FUNCTION REPLACE_CHARS : STRING(STRING_LENGTH)
VAR_INPUT
	STR : STRING(STRING_LENGTH);
	SRC : STRING;
	REP : STRING;
END_VAR
VAR
	a, b : INT;
	c: STRING(1);
	stp: INT;
END_VAR

(*
version 1.0		14. may. 2008
programmer 		hugo
tested by			hugo

REPLACE_CHARS erstezt alle character die im string src aufgeführt sind mit dem an der selben stelle im string rep gelisteten character.

*)

REPLACE_CHARS := STR;
(* make sure rep and src are of same length and length is > 0 *)
a := LEN(src);
b := LEN(rep);
IF a < b THEN
	rep := LEFT(rep, a);
ELSIF b < a THEN
	src := LEFT(src, b);
END_IF;

(* search the string and replace if necessary *)
stp := LEN(str);
FOR a := 1 TO stp DO
	c := MID(REPLACE_CHARS, 1, a);
	b := FIND(src, c);
	IF b > 0 THEN
		REPLACE_CHARS := REPLACE(REPLACE_CHARS, MID(rep, 1, b), 1, a);
	END_IF;
END_FOR;



(* revision history
hm	14. may. 2008	rev 1.0
	original version

*)

END_FUNCTION

(* stored: Version 1.1.0.1, ProductVersion 3.1.4022.7
   POU REPLACE_CHARS: Id {b34e5c6d-cd19-48ad-8d96-62a95a3ff267}, SpecialFunc None *)
